// TIA Portal V16 export
// export: Created 2021-11-12T13:33:08.1835565Z, ExportSetting WithDefaults, DisplayName Totally Integrated Automation Portal, DisplayVersion V16 Update 3, DisplayName TIA Portal Version Control Interface, DisplayVersion V16 Update 2, DisplayName TIA Portal Openness, DisplayVersion V16 Update 3, DisplayName SINAMICS Startdrive Advanced, DisplayVersion V16 Update 5, DisplayName SINAMICS Startdrive G130, G150, S120, S150, SINAMICS MV, S210, DisplayVersion V16 Update 5, DisplayName SINAMICS Startdrive G110M, G120, G120C, G120D, G120P, G115D, DisplayVersion V16 Update 5, DisplayName STEP 7 Professional, DisplayVersion V16 Update 3, DisplayName STEP 7 Safety, DisplayVersion V16, DisplayName WinCC UA Professional, DisplayVersion V16 Update 3
DATA_BLOCK "IDB_Station410"   // DB48
VERSION : 0.1
// stored: AutoNumber true, DBAccessibleFromOPCUA true, InstanceOfName Station410, InstanceOfType FB
"Station410"
   // VAR
   //    "SF_EQ01-MA01" : "STD_Drive1";
   //    "SF_EQ01-MA02" : "STD_Valve2WB";
   //    "SF_EQ01-MA03" : "STD_Valve2WB";
   //    "SF_EQ01-MA04" : "STD_Valve2WB";
   //    "SF_UC11-TA01" { S7_SetPoint := 'True'} : "STD_Siemens_G120_CU240E_2_PN";
   //    SF_Alarm1 { S7_SetPoint := 'True'} : "STD_DI_Mon";
   //    SF_Alarm2 { S7_SetPoint := 'True'} : "STD_DI_Mon";
   //    SF_Alarm3 { S7_SetPoint := 'True'} : "STD_DI_Mon";
   //    SF_Alarm4 { S7_SetPoint := 'True'} : "STD_DI_Mon";
   //    SF_Alarm5 { S7_SetPoint := 'True'} : "STD_DI_Mon";
   //    SF_Alarm6 { S7_SetPoint := 'True'} : "STD_DI_Mon";
   //    SF_Alarm7 { S7_SetPoint := 'True'} : "STD_DI_Mon";
   //    SF_Alarm8 { S7_SetPoint := 'True'} : "STD_DI_Mon";
   //    SF_Alarm9 { S7_SetPoint := 'True'} : "STD_DI_Mon";
   //    SS_Cooling : Struct
   //       LiqTemp : Real;
   //       HystMin : Real;
   //       HystMax : Real;
   //       RunPump : Bool;
   //       RegEn : Bool;
   //    END_STRUCT;
   //    SR_TmpWaterLevel : Real;
   //    SB1_PowerOk { S7_SetPoint := 'True'} : Bool;
   //    SF_TimerWaterHom { S7_SetPoint := 'True'} : TON_TIME;
   // END_VAR
BEGIN
END_DATA_BLOCK
